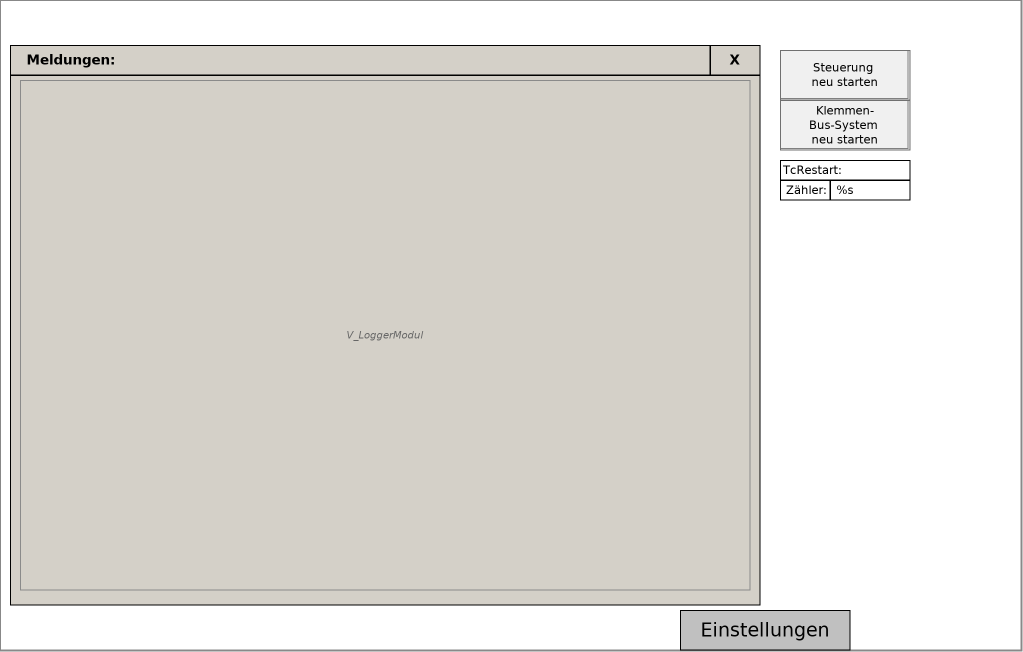
VISUALIZATION V_Logger  // 1023x652
    Frame (0,0 1021x650)
        shows V_Main_PC()
    Rectangle (680,610 170x40), "Einstellungen"
    Button (780,50 130x50), "Steuerung neu starten", invisible if: gfbSystemCX.tonStartUp.Q = 0
        OnMouseUp: change screen: V_TCReset
    Button (780,100 130x50), "Klemmen- Bus-System neu starten", invisible if: gfbSystemCX.tonStartUp.Q = 0
        OnMouseUp: change screen: V_ECReset
    Rectangle (10,75 750x530)
    Rectangle (10,45 700x30), "Meldungen:"
    Rectangle (710,45 50x30), "X"
        OnMouseClick: change screen: Previous 
    Rectangle (830,180 80x20), "%s", text variable: gfbSystemCX.nviTcRestartCnt
    Rectangle (780,160 130x20), "TcRestart:"
    Rectangle (780,180 50x20), "Zähler:"
    Frame (20,80 730x510)
        shows V_LoggerModul(fbLogger := gfbLogger)
END_VISUALIZATION

(* stored: Version 1.1.0.1, ProductVersion 3.1.4018.10
   Visu V_Logger: Id {dd8e4911-72e3-4723-b7e9-8f5e8c3f7695} *)
